FUNCTION_BLOCK AX_CYCLE (* Peroidic event generator *)
  (* Standard: 61499-1 Annex A; Description: Copyright (c) 2026 HR Agrartechnik GmbH This program and the accompanying materials are made available under the terms of the Eclipse Public License 2.0 which is available at https://www.eclipse.org/legal/epl-2.0/ SPDX-License-Identifier: EPL-2.0 *)
  (* Version 3.0, 2026-01-14, Moritz Ortmeier, HR Agrartechnik GmbH *)
  PACKAGE iec61499::events;
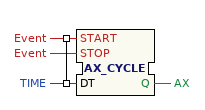
  EVENT_INPUT
    START WITH DT; (* Start the perodic generation of events *)
    STOP; (* Stop the generation of events *)
  END_EVENT
  VAR_INPUT
    DT : TIME; (* cycle time *)
  END_VAR
  PLUGS
    Q : adapter::types::unidirectional::AX;
  END_PLUGS
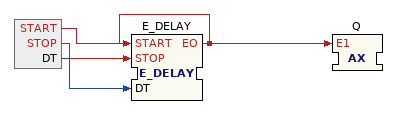
  FBS
    E_DELAY : iec61499::events::E_DELAY;
  END_FBS
  EVENT_CONNECTIONS
    START TO E_DELAY.START;
    STOP TO E_DELAY.STOP;
    E_DELAY.EO TO E_DELAY.START;
    E_DELAY.EO TO Q.E1;
  END_CONNECTIONS
  DATA_CONNECTIONS
    DT TO E_DELAY.DT;
  END_CONNECTIONS
END_FUNCTION_BLOCK
